PROGRAM MAIN
VAR
	count : DINT;
END_VAR

count := count + 1;

END_PROGRAM

(* stored: Version 1.1.0.1, ProductVersion 3.1.4026.18
   POU MAIN: Id {00000000-0000-0000-0000-0000000000a0}, SpecialFunc None *)
